FUNCTION_BLOCK FB_SlaveArm
VAR_INPUT
END_VAR
VAR_OUTPUT
END_VAR
VAR
	// arm index, from 1 to 4
	m_armIdx: INT;
	
	// grip angle
	m_gripAngle :LREAL;
	
	// joints
	m_joints :ARRAY[1..g_sJntNum] OF FB_SlaveJoint;
	
	// instrument
	m_panelOnIO AT%I*	:SINT;
	m_panelOnFlag :BOOL;
	m_instruOnIO AT%I* :SINT;
	m_instruOnFlag :BOOL;
	m_instrument : FB_Instrument;
	
	// arm cartesian data, defined in each arm origin
	m_curCartPose	:ST_Frame;
	m_curCartTwist: Vec6d;
	
	// arm joint data
	m_curMotorPos :Vec8d;
	m_curLinkPos :Vec8d;
	m_curJntPos :Vec8d;
	m_curDHJntPos :Vec6d;
	m_curGripAngle :LREAL;
	m_curJntVel :Vec8d;
	m_curJntTrq :Vec8d;
	m_cmdJntTrq :Vec8d;
	m_rawJntCurrent :Vec8d;
	m_filtJntCurrent :Vec8d;
	m_cmdJntCurrent : Vec8d;
		
	// arm dynamic data
	m_jntGravity : Vec3d;
	m_jntMassMat : Mat3d;
	
	// arm jacobian and inverse
	m_jaco : Mat6d;
	
	// simulated status
	m_simJntPos :Vec8d;
	m_simDHJntPos :Vec6d;
	m_simGripAngle :LREAL;
	m_simCartPose : ST_Frame;
	m_simJaco : Mat6d;
	m_simJacoInv :Mat6d;
	m_isSingularity:BOOL:=false;
	
	// joint position controller
	m_jntPIDCtrl :ARRAY[1..g_sJntNum] OF FB_PID;
	
END_VAR

PROPERTY armIdx : int
GET
armIdx:=m_armIdx;
END_GET
END_PROPERTY

METHOD PUBLIC calcJaco : BOOL
VAR_IN_OUT CONSTANT
	i_DHJntPos :Vec6d;
END_VAR
VAR_IN_OUT
	r_jaco :Mat6d;
END_VAR
VAR_INPUT
END_VAR

VAR
	d1, L, a, b :LREAL;
	q3:LREAL;

	c1,c2,c4,c5,c6,c7 :LREAL;
	s1,s2,s4,s5,s6,s7 :LREAL;
END_VAR
d1:=GVL_SlaveArmKinematic.g_d1;
L:=m_instrument.kinematicParameters.m_rodLength;
a:=m_instrument.kinematicParameters.m_headLength;
b:=m_instrument.kinematicParameters.m_fingerLenght;

q3:=i_DHJntPos[3];
q3:=i_DHJntPos[3];
c1:=COS(i_DHJntPos[1]);
c2:=COS(i_DHJntPos[2]);
c4:=COS(i_DHJntPos[4]);
c5:=COS(i_DHJntPos[5]);
c6:=COS(i_DHJntPos[6]);

s1:=SIN(i_DHJntPos[1]);
s2:=SIN(i_DHJntPos[2]);
s4:=SIN(i_DHJntPos[4]);
s5:=SIN(i_DHJntPos[5]);
s6:=SIN(i_DHJntPos[6]);

// jacobian with DH joints
r_jaco[1,1]:=b*(c6*(c5*(c1*s4 - c2*c4*s1) + s1*s2*s5) - s6*(c1*c4 + c2*s1*s4)) + a*(c5*(c1*s4 - c2*c4*s1) + s1*s2*s5) - L*s1*s2 + q3*s1*s2;
r_jaco[1,2]:=-c1*(a*(c2*s5 + c4*c5*s2) - L*c2 + q3*c2 + b*(c6*(c2*s5 + c4*c5*s2) + s2*s4*s6));
r_jaco[1,3]:=-c1*s2;
r_jaco[1,4]:=s1*s2*(a*(c2*s5 + c4*c5*s2) + b*(c6*(c2*s5 + c4*c5*s2) + s2*s4*s6)) - c2*(b*(c6*(c5*(c1*s4 - c2*c4*s1) + s1*s2*s5) - s6*(c1*c4 + c2*s1*s4)) + a*(c5*(c1*s4 - c2*c4*s1) + s1*s2*s5));
r_jaco[1,5]:=- (a*(c2*s5 + c4*c5*s2) + b*(c6*(c2*s5 + c4*c5*s2) + s2*s4*s6))*(c1*c4 + c2*s1*s4) - s2*s4*(b*(c6*(c5*(c1*s4 - c2*c4*s1) + s1*s2*s5) - s6*(c1*c4 + c2*s1*s4)) + a*(c5*(c1*s4 - c2*c4*s1) + s1*s2*s5));
r_jaco[1,6]:= b*(c6*(c5*(c1*s4 - c2*c4*s1) + s1*s2*s5) - s6*(c1*c4 + c2*s1*s4))*(c2*c5 - c4*s2*s5) + b*(s5*(c1*s4 - c2*c4*s1) - c5*s1*s2)*(c6*(c2*s5 + c4*c5*s2) + s2*s4*s6);


r_jaco[2,1]:=0;
r_jaco[2,2]:=c1*(a*(c5*(s1*s4 + c1*c2*c4) - c1*s2*s5) + b*(c6*(c5*(s1*s4 + c1*c2*c4) - c1*s2*s5) - s6*(c4*s1 - c1*c2*s4)) + L*c1*s2 - q3*c1*s2) - s1*(b*(c6*(c5*(c1*s4 - c2*c4*s1) + s1*s2*s5) - s6*(c1*c4 + c2*s1*s4)) + a*(c5*(c1*s4 - c2*c4*s1) + s1*s2*s5) - L*s1*s2 + q3*s1*s2);
r_jaco[2,3]:= c2;
r_jaco[2,4]:=- s1*s2*(a*(c5*(s1*s4 + c1*c2*c4) - c1*s2*s5) + b*(c6*(c5*(s1*s4 + c1*c2*c4) - c1*s2*s5) - s6*(c4*s1 - c1*c2*s4))) - c1*s2*(b*(c6*(c5*(c1*s4 - c2*c4*s1) + s1*s2*s5) - s6*(c1*c4 + c2*s1*s4)) + a*(c5*(c1*s4 - c2*c4*s1) + s1*s2*s5));
r_jaco[2,5]:=(a*(c5*(s1*s4 + c1*c2*c4) - c1*s2*s5) + b*(c6*(c5*(s1*s4 + c1*c2*c4) - c1*s2*s5) - s6*(c4*s1 - c1*c2*s4)))*(c1*c4 + c2*s1*s4) - (b*(c6*(c5*(c1*s4 - c2*c4*s1) + s1*s2*s5) - s6*(c1*c4 + c2*s1*s4)) + a*(c5*(c1*s4 - c2*c4*s1) + s1*s2*s5))*(c4*s1 - c1*c2*s4);
r_jaco[2,6]:=b*(c6*(c5*(c1*s4 - c2*c4*s1) + s1*s2*s5) - s6*(c1*c4 + c2*s1*s4))*(s5*(s1*s4 + c1*c2*c4) + c1*c5*s2) - b*(s5*(c1*s4 - c2*c4*s1) - c5*s1*s2)*(c6*(c5*(s1*s4 + c1*c2*c4) - c1*s2*s5) - s6*(c4*s1 - c1*c2*s4));

r_jaco[3,1]:=a*(c5*(s1*s4 + c1*c2*c4) - c1*s2*s5) + b*(c6*(c5*(s1*s4 + c1*c2*c4) - c1*s2*s5) - s6*(c4*s1 - c1*c2*s4)) + L*c1*s2 - q3*c1*s2;
r_jaco[3,2]:=-s1*(a*(c2*s5 + c4*c5*s2) - L*c2 + q3*c2 + b*(c6*(c2*s5 + c4*c5*s2) + s2*s4*s6));
r_jaco[3,3]:=-s1*s2;
r_jaco[3,4]:=- c2*(a*(c5*(s1*s4 + c1*c2*c4) - c1*s2*s5) + b*(c6*(c5*(s1*s4 + c1*c2*c4) - c1*s2*s5) - s6*(c4*s1 - c1*c2*s4))) - c1*s2*(a*(c2*s5 + c4*c5*s2) + b*(c6*(c2*s5 + c4*c5*s2) + s2*s4*s6));
r_jaco[3,5]:=- (a*(c2*s5 + c4*c5*s2) + b*(c6*(c2*s5 + c4*c5*s2) + s2*s4*s6))*(c4*s1 - c1*c2*s4) - s2*s4*(a*(c5*(s1*s4 + c1*c2*c4) - c1*s2*s5) + b*(c6*(c5*(s1*s4 + c1*c2*c4) - c1*s2*s5) - s6*(c4*s1 - c1*c2*s4)));
r_jaco[3,6]:=b*(c6*(c5*(s1*s4 + c1*c2*c4) - c1*s2*s5) - s6*(c4*s1 - c1*c2*s4))*(c2*c5 - c4*s2*s5) + b*(c6*(c2*s5 + c4*c5*s2) + s2*s4*s6)*(s5*(s1*s4 + c1*c2*c4) + c1*c5*s2);

r_jaco[4,1]:=0;
r_jaco[4,2]:=-s1;
r_jaco[4,3]:=0;
r_jaco[4,4]:=-c1*s2;
r_jaco[4,5]:=c1*c2*s4 - c4*s1;
r_jaco[4,6]:=s5*(s1*s4 + c1*c2*c4) + c1*c5*s2;

r_jaco[5,1]:=-1;
r_jaco[5,2]:=0;
r_jaco[5,3]:=0;
r_jaco[5,4]:=c2;
r_jaco[5,5]:=s2*s4;
r_jaco[5,6]:=c4*s2*s5 - c2*c5;

r_jaco[6,1]:=0;
r_jaco[6,2]:=c1;
r_jaco[6,3]:=0;
r_jaco[6,4]:=-s1*s2;
r_jaco[6,5]:=c1*c4 + c2*s1*s4;
r_jaco[6,6]:=c5*s1*s2 - s5*(c1*s4 - c2*c4*s1);
END_METHOD

METHOD chencPanelAndInstru : BOOL
VAR_INPUT
END_VAR
// check panel and instrument
m_panelOnFlag := panelDetect();
m_instruOnFlag := instruDetect();
IF FALSE = m_instruOnFlag THEN
	m_instrument.reset();
ELSIF InstruType_UNKNOWM = m_instrument.instruType THEN
	m_instrument.readParameters();
END_IF

m_instruOnFlag := m_instruOnFlag AND (m_instrument.instruType <> InstruType_UNKNOWM);
END_METHOD

PROPERTY cmdJntCurrent : REFERENCE TO  Vec8d
GET
cmdJntCurrent ref= m_cmdJntCurrent;
END_GET
END_PROPERTY

PROPERTY curCartPose : REFERENCE TO ST_Frame
GET
curCartPose ref=m_curCartPose;
END_GET
END_PROPERTY

PROPERTY curCartTwist : REFERENCE TO Vec6d
GET
curCartTwist ref=m_curCartTwist;
END_GET
END_PROPERTY

PROPERTY curJntPos : REFERENCE TO Vec8d
GET
curJntPos ref=m_curJntPos;
END_GET
END_PROPERTY

PROPERTY curJntTrq : REFERENCE TO Vec8d
GET
curJntTrq ref=m_curJntTrq;
END_GET
END_PROPERTY

PROPERTY curJntVel :REFERENCE TO Vec8d
GET
curJntVel ref=m_curJntVel;
END_GET
END_PROPERTY

PROPERTY curLinkPos :REFERENCE TO Vec8d
GET
curLinkPos ref=m_curLinkPos;
END_GET
END_PROPERTY

PROPERTY curMotorPos : REFERENCE TO  Vec8d
GET
curMotorPos ref=m_curMotorPos;
END_GET
END_PROPERTY

METHOD PUBLIC enable : BOOL
VAR_IN_OUT CONSTANT
	i_jntIdx :Vec8i;
END_VAR
VAR
	i :INT ;
END_VAR
FOR i:=1 TO g_sJntNum DO
	IF 1= i_jntIdx[i] THEN
		m_joints[i].enable();
	ELSE
		m_joints[i].disable();
	END_IF
END_FOR
END_METHOD

PROPERTY filtJntCurrent :REFERENCE TO Vec8d
GET
filtJntCurrent ref= m_filtJntCurrent;
END_GET
END_PROPERTY

// from active joint position to cartesian pose in arm origin
METHOD PROTECTED forwardKinematic : BOOL
VAR_IN_OUT CONSTANT
	i_DHJntPos :Vec6d;
END_VAR
VAR_IN_OUT
	r_cartPose :ST_Frame;
	r_gripAngle : LREAL;
END_VAR
VAR
	d1, L, a, b :LREAL;
	q3 :LREAL;

	c1,c2,c4,c5,c6,c7 :LREAL;
	s1,s2,s4,s5,s6,s7 :LREAL;

END_VAR

d1:=GVL_SlaveArmKinematic.g_d1;
L:=m_instrument.kinematicParameters.m_rodLength;
a:=m_instrument.kinematicParameters.m_headLength;
b:=m_instrument.kinematicParameters.m_fingerLenght;

q3:=i_DHJntPos[3];
c1:=COS(i_DHJntPos[1]);
c2:=COS(i_DHJntPos[2]);
c4:=COS(i_DHJntPos[4]);
c5:=COS(i_DHJntPos[5]);
c6:=COS(i_DHJntPos[6]);

s1:=SIN(i_DHJntPos[1]);
s2:=SIN(i_DHJntPos[2]);
s4:=SIN(i_DHJntPos[4]);
s5:=SIN(i_DHJntPos[5]);
s6:=SIN(i_DHJntPos[6]);


// cartesian pose frame
r_cartPose.m_pos[1]:=a*(c5*(s1*s4 + c1*c2*c4) - c1*s2*s5) + b*(c6*(c5*(s1*s4 + c1*c2*c4) - c1*s2*s5) - s6*(c4*s1 - c1*c2*s4)) + L*c1*s2 - q3*c1*s2;
r_cartPose.m_pos[2]:=a*(c2*s5 + c4*c5*s2) - d1 - L*c2 + q3*c2 + b*(c6*(c2*s5 + c4*c5*s2) + s2*s4*s6);
r_cartPose.m_pos[3]:=L*s1*s2 - a*(c5*(c1*s4 - c2*c4*s1) + s1*s2*s5) - b*(c6*(c5*(c1*s4 - c2*c4*s1) + s1*s2*s5) - s6*(c1*c4 + c2*s1*s4)) - q3*s1*s2;

r_cartPose.m_rot[1,1]:= c6*(c5*(s1*s4 + c1*c2*c4) - c1*s2*s5) - s6*(c4*s1 - c1*c2*s4);
r_cartPose.m_rot[2,1]:=c6*(c2*s5 + c4*c5*s2) + s2*s4*s6;
r_cartPose.m_rot[3,1]:=s6*(c1*c4 + c2*s1*s4) - c6*(c5*(c1*s4 - c2*c4*s1) + s1*s2*s5);

r_cartPose.m_rot[1,2]:=- s6*(c5*(s1*s4 + c1*c2*c4) - c1*s2*s5) - c6*(c4*s1 - c1*c2*s4);
r_cartPose.m_rot[2,2]:=c6*s2*s4 - s6*(c2*s5 + c4*c5*s2);
r_cartPose.m_rot[3,2]:=s6*(c5*(c1*s4 - c2*c4*s1) + s1*s2*s5) + c6*(c1*c4 + c2*s1*s4);

r_cartPose.m_rot[1,3]:= s5*(s1*s4 + c1*c2*c4) + c1*c5*s2;
r_cartPose.m_rot[2,3]:= c4*s2*s5 - c2*c5;
r_cartPose.m_rot[3,3]:=c5*s1*s2 - s5*(c1*s4 - c2*c4*s1);
END_METHOD

PROPERTY gripAngle : LREAL
GET
gripAngle:=m_gripAngle;
END_GET
END_PROPERTY

METHOD PUBLIC init : BOOL
VAR_INPUT
	i_armIdx:INT;
END_VAR
VAR 
	i :INT ;
	currentRatioMotor2Jnt: LREAL;
END_VAR
// arm statues init
m_armIdx:=i_armIdx;
m_gripAngle:=0;

// joint init
FOR i:=1 TO g_sJntNum DO
	m_joints[i].init(m_armIdx, i);
END_FOR

// init joint encoder and position calculation
initJntPos();

// joint controller init
FOR i:=1 TO g_sJntNum DO 
	currentRatioMotor2Jnt:=GVL_SlaveMotorParameters.g_motorTrqConst[i]*GVL_SlaveMotorParameters.g_motorReduction[i]/1000;
	m_jntPIDCtrl[i].init(g_slaveArmCtrlCycleTime,GVL_slaveControlParameters.g_posKp[i],GVL_slaveControlParameters.g_posKd[i],
		GVL_slaveControlParameters.g_posKi[i], GVL_slaveControlParameters.g_posKiLimit[i]* currentRatioMotor2Jnt,
		GVL_slaveControlParameters.g_posCtrlLimit[i]*currentRatioMotor2Jnt);
END_FOR

// compute current status
updateStatus();
END_METHOD

METHOD initJntPos : BOOL
VAR_INPUT
END_VAR
VAR
	i:INT ;
END_VAR
// joint init
FOR i:=1 TO g_sJntNum DO
	m_joints[i].initJntPos();
END_FOR
END_METHOD

// check if instrument is on
METHOD instruDetect : BOOL
VAR_INPUT
END_VAR
//TODO
END_METHOD

PROPERTY instrument : REFERENCE TO FB_Instrument
GET
instrument REF=m_instrument;
END_GET
END_PROPERTY

PROPERTY instruOn : bool
GET
instruOn:=m_instruOnFlag;
END_GET
END_PROPERTY

METHOD PUBLIC isEnabled : BOOL
VAR_IN_OUT CONSTANT
	i_jntIdx :Vec8i;
END_VAR
VAR
	i :INT ;
END_VAR
isEnabled := TRUE;
FOR i:=1 TO g_sJntNum DO
	IF 1= i_jntIdx[i] THEN
		isEnabled :=  (m_joints[i].isEnabled() AND isEnabled);
	END_IF
END_FOR
END_METHOD

PROPERTY isSingurality : bool
GET
isSingurality:=m_isSingularity;
END_GET
END_PROPERTY

PROPERTY jaco :REFERENCE TO Mat6d
GET
jaco := m_jaco;
END_GET
END_PROPERTY

PROPERTY jntGravity :REFERENCE TO Vec3d
GET
jntGravity:=m_jntGravity;
END_GET
END_PROPERTY

PROPERTY PUBLIC massMat :REFERENCE TO Mat3d
GET
massMat :=m_jntMassMat;
END_GET
END_PROPERTY

// check if panel is on
METHOD panelDetect : BOOL
VAR_INPUT
END_VAR
// TODO
END_METHOD

PROPERTY panelOn : bool
GET
panelOn :=m_panelOnFlag;
END_GET
END_PROPERTY

PROPERTY rawJntCurrent :REFERENCE TO Vec8d
GET
rawJntCurrent:=m_rawJntCurrent;
END_GET
END_PROPERTY

METHOD readInstruInfo : BOOL
VAR_INPUT
END_VAR
m_instrument.readParameters();
END_METHOD

PROPERTY simCartPose :REFERENCE TO ST_Frame
GET
simCartPose:=m_simCartPose;
END_GET
END_PROPERTY

PROPERTY simJaco :REFERENCE TO mat6d
GET
simJaco:=m_simJaco;
END_GET
END_PROPERTY

// update joints control command
METHOD PUBLIC updateCmds : BOOL
VAR_IN_OUT CONSTANT
	i_armCtrlCmd : ST_SlaveArmCtrlCmds;
END_VAR
VAR
	i:INT;
END_VAR
m_cmdJntTrq:=i_armCtrlCmd.m_cmdJntTrq;
m_simJntPos:=i_armCtrlCmd.m_cmdJntPos;

// update simulated master arm
updateSimStatus();

// enable/disable joints
enable(i_armCtrlCmd.m_jntEnableFlag);

// position/torque control
FOR i:=1 TO g_sJntNum DO 
	IF i_armCtrlCmd.m_jntOPMode[i]=DriverOPMode_PosTrq THEN
		// position controller and gravity feedforward
		m_cmdJntTrq[i]:=m_jntPIDCtrl[i].run(i_armCtrlCmd.m_cmdJntPos[i],m_curJntPos[i],i_armCtrlCmd.m_cmdJntVel[i],m_curJntVel[i]);
		m_cmdJntTrq[i]:=m_cmdJntTrq[i]+m_jntGravity[i];
		m_joints[i].updateCmds(DriverOPMode_Trq,i_armCtrlCmd.m_cmdJntPos[i],m_cmdJntTrq[i]);
	ELSIF i_armCtrlCmd.m_jntOPMode[i]=DriverOPMode_Trq THEN
		// gravity feedforward
		m_cmdJntTrq[i]:=m_cmdJntTrq[i]+m_jntGravity[i];
		m_joints[i].updateCmds(DriverOPMode_Trq,i_armCtrlCmd.m_cmdJntPos[i],m_cmdJntTrq[i]);
	ELSE
		m_jntPIDCtrl[i].reset();
		m_cmdJntTrq[i]:=0;
		m_joints[i].updateCmds(DriverOPMode_Pos,i_armCtrlCmd.m_cmdJntPos[i],m_cmdJntTrq[i]);
	END_IF
	
END_FOR
END_METHOD

METHOD PUBLIC updateDyna : BOOL
VAR_IN_out constant
	slaveDynaData : ST_SlaveDynaData;
END_VAR
m_jntMassMat:=slaveDynaData.m_massMat[m_armIdx];
m_jntGravity:=slaveDynaData.m_gravity[m_armIdx];
END_METHOD

METHOD PUBLIC updateSimStatus : BOOL
VAR_INPUT
END_VAR
//IF m_instrument.ready THEN
	// instrument kinematic
	m_instrument.instruFK(m_simJntPos, m_simDHJntPos, m_simGripAngle);

	// simulated cartesion pose 
	forwardKinematic(m_simDHJntPos,m_simCartPose,m_simGripAngle);
	
	// simulated jacobian
	calcJaco(m_simDHJntPos,m_simJaco);
	m_isSingularity:=NOT(invMat6(m_simJaco, m_simJacoInv));
//END_IF
END_METHOD

// update arm status, including kinematic and dynamic
METHOD PUBLIC updateStatus : BOOL
VAR_INPUT
END_VAR
VAR 
	i,j:INT;
END_VAR
// update joint data
FOR i:=1 TO g_sJntNum DO
	m_joints[i].updateStatus();
END_FOR

// check panel and instrument
chencPanelAndInstru();

// get joint data
FOR i:=1 TO g_sJntNum DO
	m_curMotorPos[i]:=m_joints[i].motorPos;
	m_curLinkPos[i]:=m_joints[i].linkPos;
	m_curJntPos[i]:=m_joints[i].jntPos;
	m_curJntVel[i]:=m_joints[i].jntVel;
	m_curJntTrq[i]:=m_joints[i].jntTrq;
	m_rawJntCurrent[i]:=m_joints[i].rawCurrent;
	m_filtJntCurrent[i]:=m_joints[i].filtCurrent;
	m_cmdJntCurrent[i]:=m_joints[i].cmdCurrent;
END_FOR 

// only update carteisn data when instrument is ready
//IF m_instrument.ready THEN
	
	// instrument kinematic
	m_instrument.instruFK(m_curJntPos, m_curDHJntPos, m_curGripAngle);

	// cartesion pose
	forwardKinematic(m_curDHJntPos,m_curCartPose,m_gripAngle);
	
	// jacobian
	calcJaco(m_curDHJntPos,m_jaco);
	
	// cartesian twist
//END_IF
END_METHOD

END_FUNCTION_BLOCK

(* stored: Version 1.1.0.1, ProductVersion 3.1.4024.12
   POU FB_SlaveArm: Id {623926f8-06e2-46b6-bb1f-baa6bc16e9cb}, SpecialFunc None
   Folder property: Id {4aa1799c-1556-4bc1-a713-06f14faa00f1}
   Property armIdx: Id {1bcadfc3-0a4f-4bee-a1a7-b6d4d3a1eb58}
   Get Get: Id {198387ec-2e24-42e6-b0c2-2f769705d46f}
   Method calcJaco: Id {1172e5e4-b7f2-4690-a821-6304414cea84}
   Method chencPanelAndInstru: Id {613633aa-f5bc-4224-95e6-e974a90f8e6a}
   Property cmdJntCurrent: Id {cbd7aa84-e545-47b8-bdc5-960aa8409c91}
   Get Get: Id {12be56c2-8b79-47d6-b1f2-86b8e0a5f91a}
   Property curCartPose: Id {d18be23c-99e5-435e-8688-90e0fb3be9ca}
   Get Get: Id {013b03f6-adb7-4855-b0fe-353f77f67094}
   Property curCartTwist: Id {e4b7010c-887c-41fa-8766-1a9192e9d06a}
   Get Get: Id {b7c89bf7-90fc-4841-be25-e467b1918b68}
   Property curJntPos: Id {d72c054a-bae9-44cb-97ff-fe7c76c53cb8}
   Get Get: Id {332d5297-fb56-44bd-a751-714464e0813c}
   Property curJntTrq: Id {8c78ba58-302c-4844-9d36-e487700a0e19}
   Get Get: Id {1767bffb-cddd-4133-ad6f-5125f86340af}
   Property curJntVel: Id {904c68d5-30c9-4ed3-b3c5-6bcd345bcd5a}
   Get Get: Id {0a508621-c577-4d50-8cc3-bd8133f79f72}
   Property curLinkPos: Id {3725bf51-2c50-4574-b2a7-e2af9fd4da29}
   Get Get: Id {cff7c92f-5276-4a58-b7ca-f6248868b409}
   Property curMotorPos: Id {ad9d9e24-10f4-4dc4-b0d2-86517dead53b}
   Get Get: Id {bc557e46-3cdd-47ba-9e7f-cf7525f3969d}
   Method enable: Id {596f2892-08b6-4851-84d5-1537c558264e}
   Property filtJntCurrent: Id {1f5e4c97-ef8c-417a-90ec-656c048c0e4f}
   Get Get: Id {34ea0c3d-b0bc-4adb-bbb3-f4ab6640a7ff}
   Method forwardKinematic: Id {182b544f-f7c4-475e-8af7-8c07aa230234}
   Property gripAngle: Id {5187a911-df75-4b56-8b45-38142d9b24de}
   Get Get: Id {871729fd-1ba1-4906-aec3-7d572491feb2}
   Method init: Id {d7bcc040-c32e-4455-ab43-70de0dc2919e}
   Method initJntPos: Id {56ee4071-fcb1-4318-b1b9-837ea21e1627}
   Method instruDetect: Id {5f3a6988-31d6-440d-837a-fcdd94d64d1d}
   Property instrument: Id {ef5d0758-d499-4e04-a177-87950f9a716b}
   Get Get: Id {3a5249de-ec45-4e88-a302-3df6650a3ff5}
   Property instruOn: Id {4486d0c9-79b0-4e6c-acfb-23ca16ba44f5}
   Get Get: Id {daa69233-49df-439c-8476-605873205ebf}
   Method isEnabled: Id {00a67cf8-62b1-4004-a2ca-9469bb0f3cab}
   Property isSingurality: Id {da3c3ca8-d645-443c-af9d-86ff4ca01cff}
   Get Get: Id {69dc0611-36d4-4919-91ba-cfdefe53366b}
   Property jaco: Id {2c2ce445-b511-4254-9c8e-e5667e1b6bdb}
   Get Get: Id {27a6e900-c6e6-40c0-aa03-4dc0d1214554}
   Property jntGravity: Id {72dbb3a4-f37f-4edd-afb1-2190cd1f62fc}
   Get Get: Id {5c8a2ae5-eaad-400d-b638-ec46a75b5ccb}
   Property massMat: Id {c4fbf6a1-1d71-4f80-9bfa-395c19261a6f}
   Get Get: Id {b8079ba8-3835-474b-9d8e-6afd86dc6a9b}
   Method panelDetect: Id {2a3a3fa1-2046-472e-b693-4c66bf1a37b0}
   Property panelOn: Id {38ffa1da-012d-4dbc-ad5b-314577ed285b}
   Get Get: Id {b8c5f533-4196-44c4-9a48-01cc1ca3c250}
   Property rawJntCurrent: Id {f1221838-7bcd-4d84-b9f8-7dc96a864978}
   Get Get: Id {23a8503d-4e33-47db-b530-039bdd0d530f}
   Method readInstruInfo: Id {67d65d43-e812-409d-9cd7-51d04d997421}
   Property simCartPose: Id {6426ffc4-f74f-4984-ac32-a9f9d8b8c8ca}
   Get Get: Id {a61bb7de-a7ad-4b34-8063-e53c825d0db4}
   Property simJaco: Id {0fa24ffb-bfb3-496c-82de-08842f53e6e4}
   Get Get: Id {35c7dda2-112e-4042-99cd-4eac5d67ff5e}
   Method updateCmds: Id {4f271d3a-4b2b-4f85-986e-f8fdffb5994c}
   Method updateDyna: Id {02de28e3-c8a7-46cf-834a-5bf048b5e039}
   Method updateSimStatus: Id {f15ad7c2-6655-4b50-9555-9aa968e8753f}
   Method updateStatus: Id {21b3fe9a-0eba-4313-bb9a-33b1f0038771} *)
